FUNCTION_BLOCK TcoDigitalActuator EXTENDS TcoCore.TcoComponent
VAR_IN_OUT
	inoSignal : BOOL;
END_VAR

VAR
	_signal : BOOL;
	_adr : ULINT;
END_VAR

IF(__ISVALIDREF(inoSignal)) THEN
	 inoSignal := _signal;
	_adr := ADR(inoSignal);
END_IF;

METHOD FB_init : BOOL
VAR_INPUT
	bInitRetains : BOOL; // if TRUE, the retain variables are initialized (warm start / cold start)
	bInCopyCode : BOOL;  // if TRUE, the instance afterwards gets moved into the copy code (online change)
	Parent : ITcoObject;
END_VAR
END_METHOD

{attribute 'monitoring' := 'variable'}
PROPERTY IsFalse : BOOL
GET
IsFalse := NOT _signal;
Messenger.Info('Expecting `negative` signal');
END_GET
END_PROPERTY

{attribute 'monitoring' := 'variable'}
PROPERTY IsTrue : BOOL
GET
IsTrue := _signal;
Messenger.Info('Expecting `positive` signal');
END_GET
END_PROPERTY

METHOD Reset : BOOL
Messenger.Trace('<#Reseting signal (off/false)#>');
_signal := FALSE;
Reset := TRUE;
END_METHOD

(*~
	<docu>
		<summary>
			Restores this instance to the Ready state. Can be called explicitly or from within one of the restore mechanisms.	
		</summary>			
	</docu>	
~*)
METHOD  Restore : ITcoRestorable
// No implementation needed for this componet.
END_METHOD

(*~
	<docu>
		<summary>
		    Custom service (manual, maintenance) logic.
			This method must be implemented in derived class.
		</summary>			
	</docu>	
~*)
METHOD PROTECTED  ServiceMode
END_METHOD

METHOD PUBLIC Set : BOOL
Messenger.Trace('<#Setting signal (on/true)#>');
_signal := TRUE;
Set := TRUE;
END_METHOD

END_FUNCTION_BLOCK

(* stored: Version 1.1.0.1, ProductVersion 3.1.4024.6
   POU TcoDigitalActuator: Id {a94c677a-ea37-0c4d-2eda-a26d576606a9}, SpecialFunc None
   Method FB_init: Id {3d495706-c76b-095e-389f-7ba6c1dae3a7}
   Property IsFalse: Id {d6d0da98-c1ac-0a37-21f7-b9013b7a9347}
   Get Get: Id {efc004b0-702d-0b7b-3249-c46f50548bad}
   Property IsTrue: Id {bfef7889-549c-0855-3e52-92d7219d024a}
   Get Get: Id {97720d5a-b86c-0dbf-0b94-b72b60d909a7}
   Method Reset: Id {8d9a1541-7fde-0939-1d52-c21f46132ca4}
   Method Restore: Id {28f0fb71-aa8a-0f79-0fa8-867a06c586ce}
   Method ServiceMode: Id {370c3428-cc83-04b9-0717-e7260a4027a0}
   Method Set: Id {83e12c95-7ea1-0597-1f2a-882d3fad52b0} *)
